// TwinCAT 3 PLC project PLC_SafetyInterlocks
// ProgramVersion: 3.1.4024.0
// libraries:
//   Tc2_Standard, * (Beckhoff Automation GmbH)
//   Tc2_System, * (Beckhoff Automation GmbH)
//   Tc3_Module, * (Beckhoff Automation GmbH)
// project tree:
//   DUTs/ E_SafeSequenceState.TcDUT, FB_EStop.TcPOU
//   / PlcTask.TcTTO
//   POUs/ MAIN.TcPOU
// real-time tasks:
//   TASK PlcTask: cycle T#10ms, priority 20, ADS port 350

CONFIGURATION PLC_SafetyInterlocks
    RESOURCE PLC ON TwinCAT3
        TASK PlcTask(INTERVAL := T#10ms, PRIORITY := 20);
        PROGRAM MAIN WITH PlcTask : MAIN;
    END_RESOURCE
END_CONFIGURATION

// ---- DUTs/E_SafeSequenceState.TcDUT
{attribute 'qualified_only'}
{attribute 'strict'}
TYPE E_SafeSequenceState :
(
	IDLE := 0,
	RUNNING := 1,
	FAULT := 2,
	RESET_PENDING := 3
);
END_TYPE

// ---- POUs/MAIN.TcPOU
PROGRAM MAIN
VAR
	eState : E_SafeSequenceState := E_SafeSequenceState.IDLE;
	bStartButton : BOOL;
	bEStopRaw : BOOL;
	bResetButton : BOOL;
	bConveyorRun : BOOL;
	fbEStop : FB_EStop;
END_VAR

fbEStop(bEStopRaw := bEStopRaw, bResetButton := bResetButton);

IF fbEStop.bFaultActive THEN
	eState := E_SafeSequenceState.FAULT;
END_IF

CASE eState OF
	E_SafeSequenceState.IDLE:
		bConveyorRun := FALSE;
		IF bStartButton THEN
			eState := E_SafeSequenceState.RUNNING;
		END_IF
		
	E_SafeSequenceState.RUNNING:
		bConveyorRun := TRUE;
		
	E_SafeSequenceState.FAULT:
		bConveyorRun := FALSE;
		IF NOT fbEStop.bFaultActive THEN
			eState := E_SafeSequenceState.IDLE;
		END_IF
END_CASE

END_PROGRAM

// ---- DUTs/FB_EStop.TcPOU
FUNCTION_BLOCK FB_EStop
VAR_INPUT
	bEStopRaw : BOOL; // TRUE = e=stop physically pressed
	bResetButton : BOOL; // operator reset after clearing fault
END_VAR
VAR_OUTPUT
	bFaultActive : BOOL; // latched fault state
END_VAR
VAR
	rTrigEStop : R_TRIG;
	rTrigReset : R_TRIG;
END_VAR

rtrigEstop(CLK := bEStopRaw);
rtrigReset(CLK := bResetButton);

IF rtrigEStop.Q THEN
	bFaultActive := TRUE;
END_IF

IF rtrigReset.Q AND NOT bEStopRaw THEN
	bFaultActive := FALSE;
END_IF

END_FUNCTION_BLOCK
